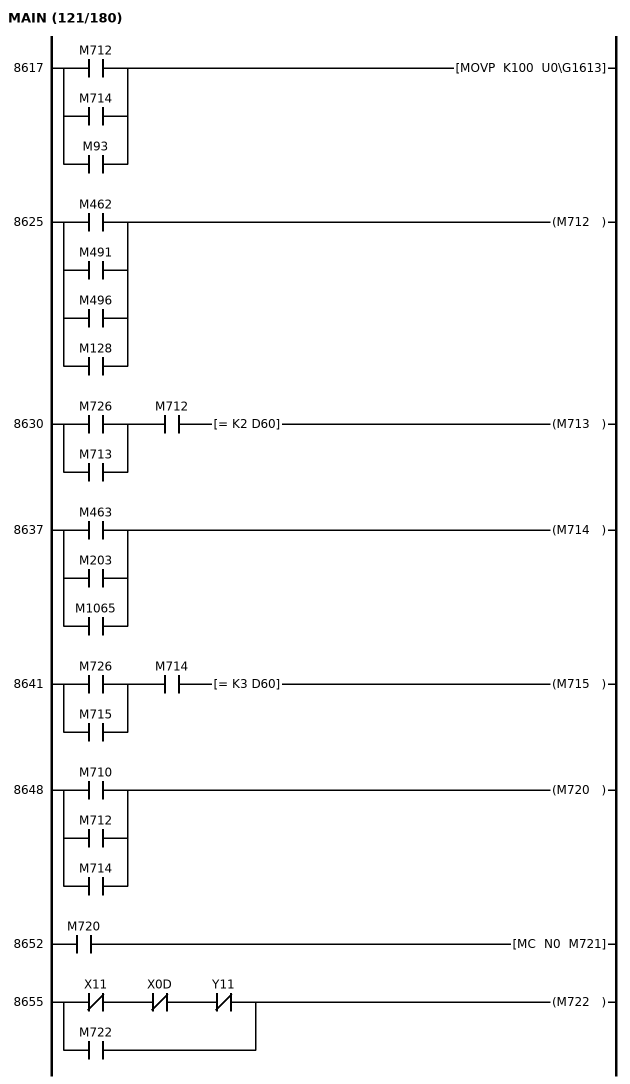
[picture p120: ladder of MAIN, rungs at steps 8617 to 8655]
8617  LD      M712
      OR      M714
      OR      M93
      MOVP    K100 U0\G1613
8625  LD      M462
      OR      M491
      OR      M496
      OR      M128
      OUT     M712
8630  LD      M726
      OR      M713
      AND     M712
      AND=    K2 D60
      OUT     M713
8637  LD      M463
      OR      M203
      OR      M1065
      OUT     M714
8641  LD      M726
      OR      M715
      AND     M714
      AND=    K3 D60
      OUT     M715
8648  LD      M710
      OR      M712
      OR      M714
      OUT     M720
8652  LD      M720
      MC      N0 M721
8655  LDI     X11
      ANI     X0D
      ANI     Y11
      OR      M722
      OUT     M722
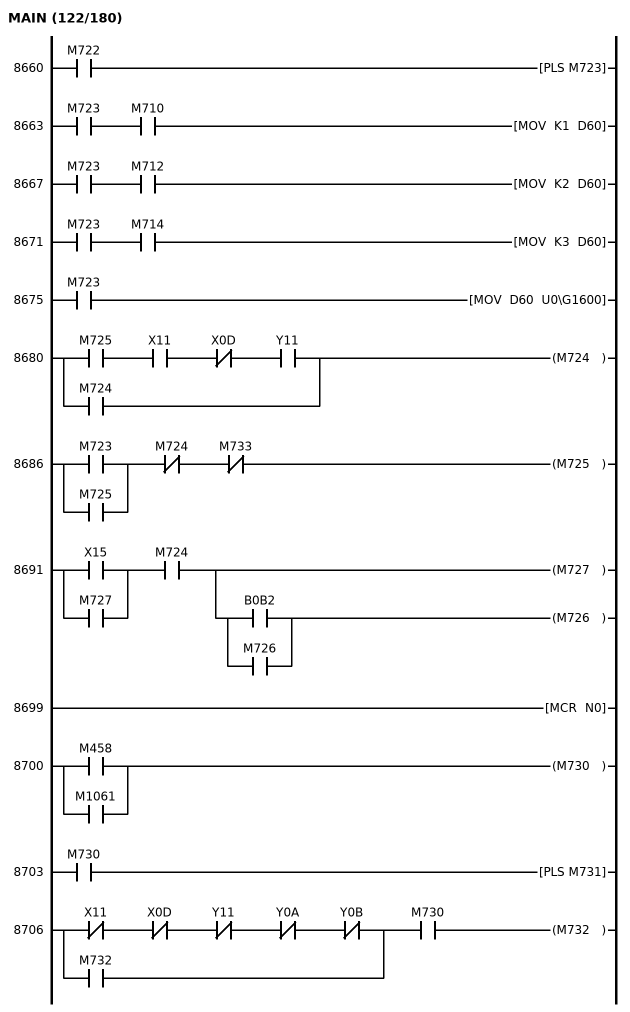
8660  LD      M722
      PLS     M723
8663  LD      M723
      AND     M710
      MOV     K1 D60
8667  LD      M723
      AND     M712
      MOV     K2 D60
8671  LD      M723
      AND     M714
      MOV     K3 D60
8675  LD      M723
      MOV     D60 U0\G1600
8680  LD      M725
      AND     X11
      ANI     X0D
      AND     Y11
      OR      M724
      OUT     M724
8686  LD      M723
      OR      M725
      ANI     M724
      ANI     M733
      OUT     M725
8691  LD      X15
      OR      M727
      AND     M724
      OUT     M727
      LD      B0B2
      OR      M726
      ANB
      OUT     M726
8699  MCR     N0
8700  LD      M458
      OR      M1061
      OUT     M730
8703  LD      M730
      PLS     M731
8706  LDI     X11
      ANI     X0D
      ANI     Y11
      ANI     Y0A
      ANI     Y0B
      OR      M732
      AND     M730
      OUT     M732
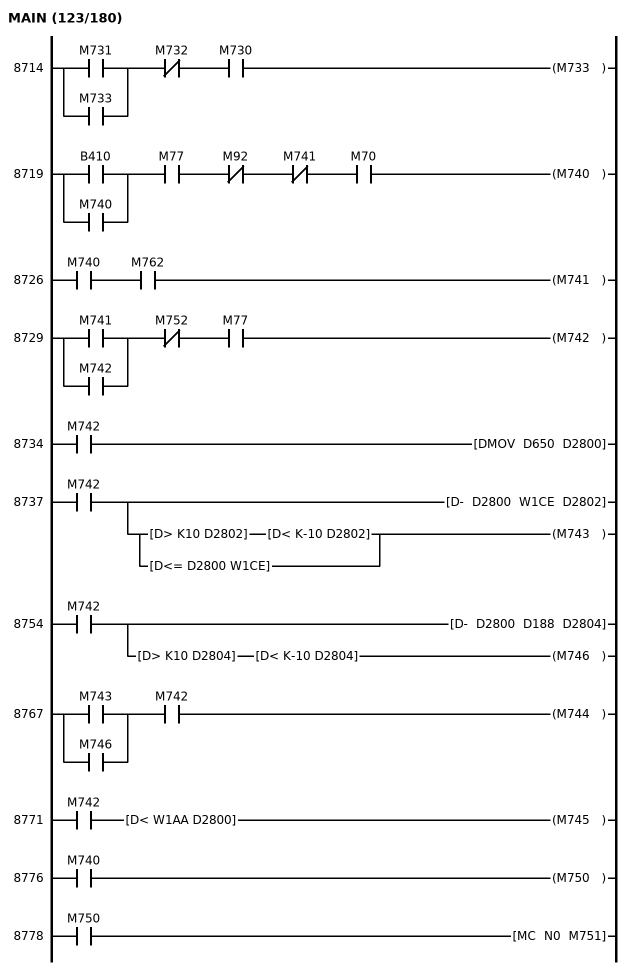
8714  LD      M731
      OR      M733
      ANI     M732
      AND     M730
      OUT     M733
8719  LD      B410
      OR      M740
      AND     M77
      ANI     M92
      ANI     M741
      AND     M70
      OUT     M740
8726  LD      M740
      AND     M762
      OUT     M741
8729  LD      M741
      OR      M742
      ANI     M752
      AND     M77
      OUT     M742
8734  LD      M742
      DMOV    D650 D2800
8737  LD      M742
      D-      D2800 W1CE D2802
      LDD>    K10 D2802
      ANDD<   K-10 D2802
      ORD<=   D2800 W1CE
      ANB
      OUT     M743
8754  LD      M742
      D-      D2800 D188 D2804
      ANDD>   K10 D2804
      ANDD<   K-10 D2804
      OUT     M746
8767  LD      M743
      OR      M746
      AND     M742
      OUT     M744
8771  LD      M742
      ANDD<   W1AA D2800
      OUT     M745
8776  LD      M740
      OUT     M750
8778  LD      M750
      MC      N0 M751
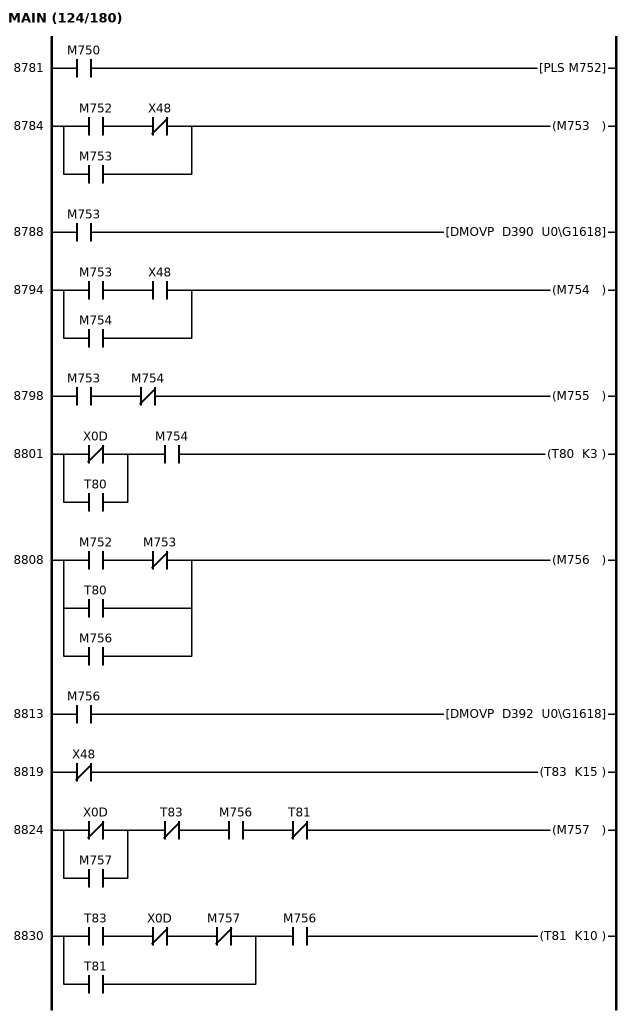
8781  LD      M750
      PLS     M752
8784  LD      M752
      ANI     X48
      OR      M753
      OUT     M753
8788  LD      M753
      DMOVP   D390 U0\G1618
8794  LD      M753
      AND     X48
      OR      M754
      OUT     M754
8798  LD      M753
      ANI     M754
      OUT     M755
8801  LDI     X0D
      OR      T80
      AND     M754
      OUT     T80 K3
8808  LD      M752
      ANI     M753
      OR      T80
      OR      M756
      OUT     M756
8813  LD      M756
      DMOVP   D392 U0\G1618
8819  LDI     X48
      OUT     T83 K15
8824  LDI     X0D
      OR      M757
      ANI     T83
      AND     M756
      ANI     T81
      OUT     M757
8830  LD      T83
      ANI     X0D
      ANI     M757
      OR      T81
      AND     M756
      OUT     T81 K10
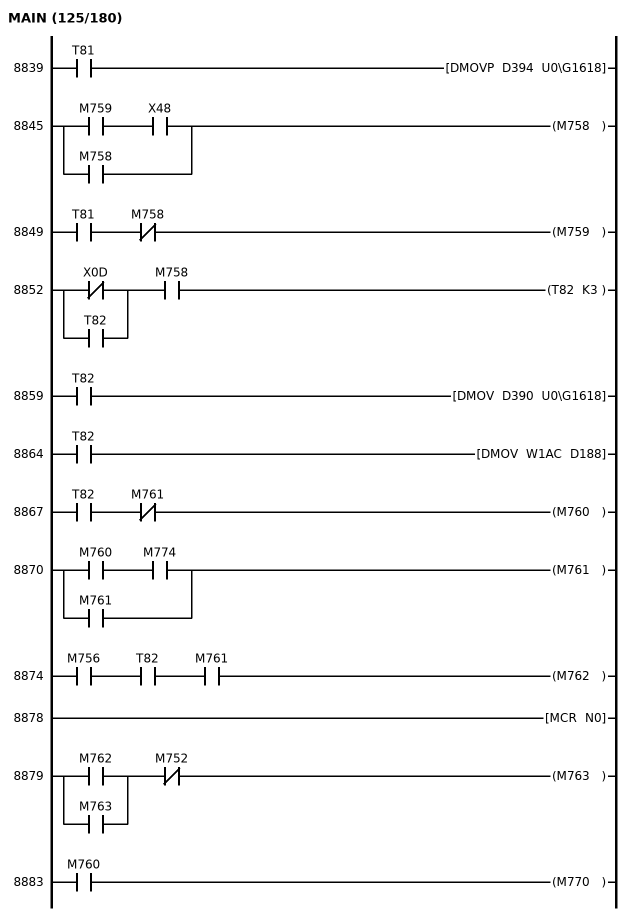
8839  LD      T81
      DMOVP   D394 U0\G1618
8845  LD      M759
      AND     X48
      OR      M758
      OUT     M758
8849  LD      T81
      ANI     M758
      OUT     M759
8852  LDI     X0D
      OR      T82
      AND     M758
      OUT     T82 K3
8859  LD      T82
      DMOV    D390 U0\G1618
8864  LD      T82
      DMOV    W1AC D188
8867  LD      T82
      ANI     M761
      OUT     M760
8870  LD      M760
      AND     M774
      OR      M761
      OUT     M761
8874  LD      M756
      AND     T82
      AND     M761
      OUT     M762
8878  MCR     N0
8879  LD      M762
      OR      M763
      ANI     M752
      OUT     M763
8883  LD      M760
      OUT     M770
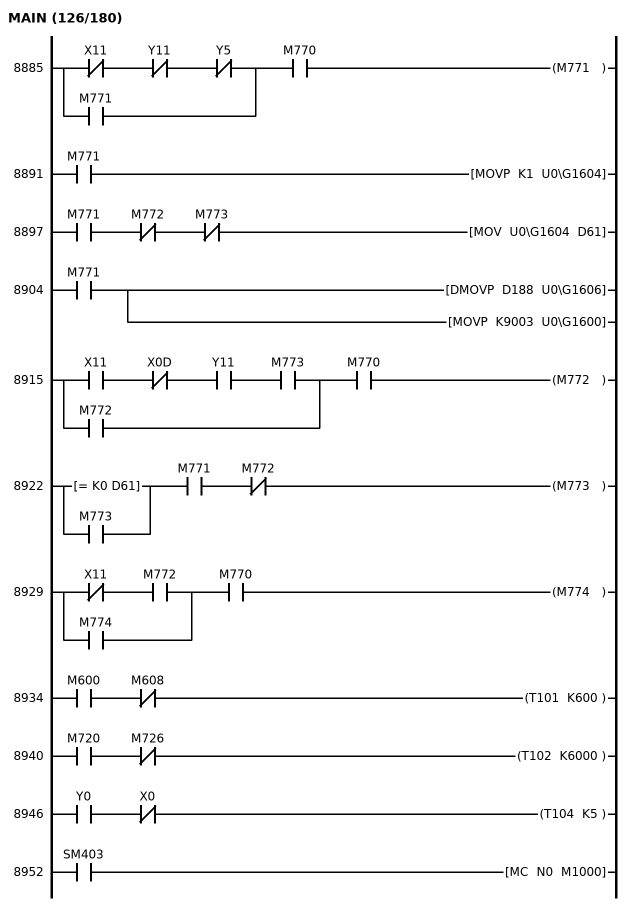
8885  LDI     X11
      ANI     Y11
      ANI     Y5
      OR      M771
      AND     M770
      OUT     M771
8891  LD      M771
      MOVP    K1 U0\G1604
8897  LD      M771
      ANI     M772
      ANI     M773
      MOV     U0\G1604 D61
8904  LD      M771
      DMOVP   D188 U0\G1606
      MOVP    K9003 U0\G1600
8915  LD      X11
      ANI     X0D
      AND     Y11
      AND     M773
      OR      M772
      AND     M770
      OUT     M772
8922  LD=     K0 D61
      OR      M773
      AND     M771
      ANI     M772
      OUT     M773
8929  LDI     X11
      AND     M772
      OR      M774
      AND     M770
      OUT     M774
8934  LD      M600
      ANI     M608
      OUT     T101 K600
8940  LD      M720
      ANI     M726
      OUT     T102 K6000
8946  LD      Y0
      ANI     X0
      OUT     T104 K5
8952  LD      SM403
      MC      N0 M1000
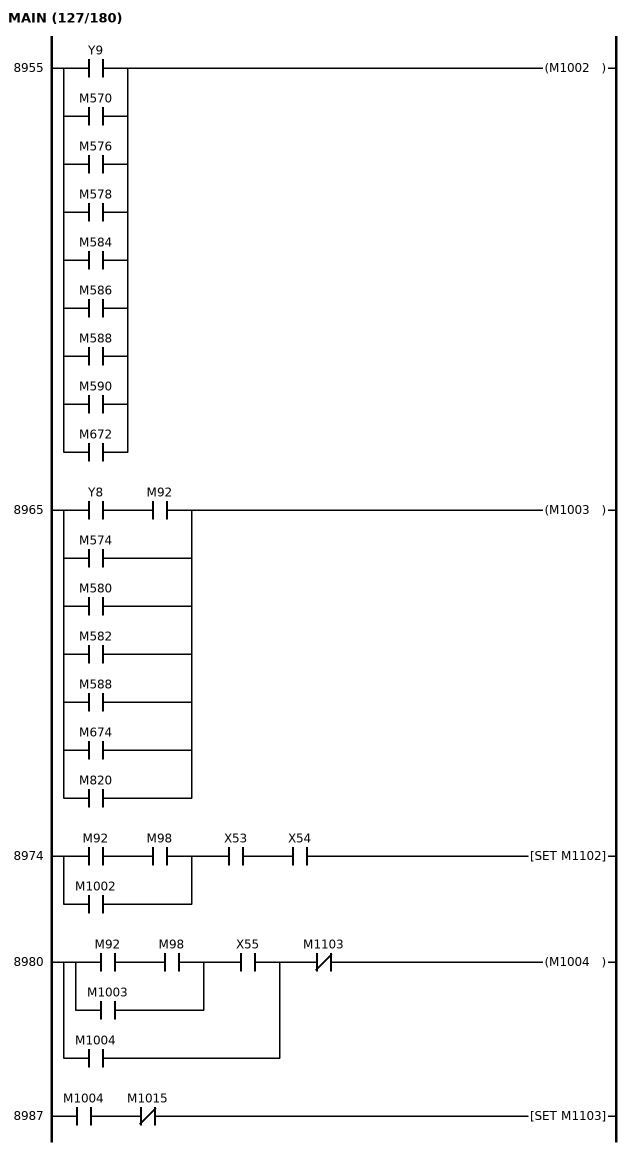
8955  LD      Y9
      OR      M570
      OR      M576
      OR      M578
      OR      M584
      OR      M586
      OR      M588
      OR      M590
      OR      M672
      OUT     M1002
8965  LD      Y8
      AND     M92
      OR      M574
      OR      M580
      OR      M582
      OR      M588
      OR      M674
      OR      M820
      OUT     M1003
8974  LD      M92
      AND     M98
      OR      M1002
      AND     X53
      AND     X54
      SET     M1102
8980  LD      M92
      AND     M98
      OR      M1003
      AND     X55
      OR      M1004
      ANI     M1103
      OUT     M1004
8987  LD      M1004
      ANI     M1015
      SET     M1103
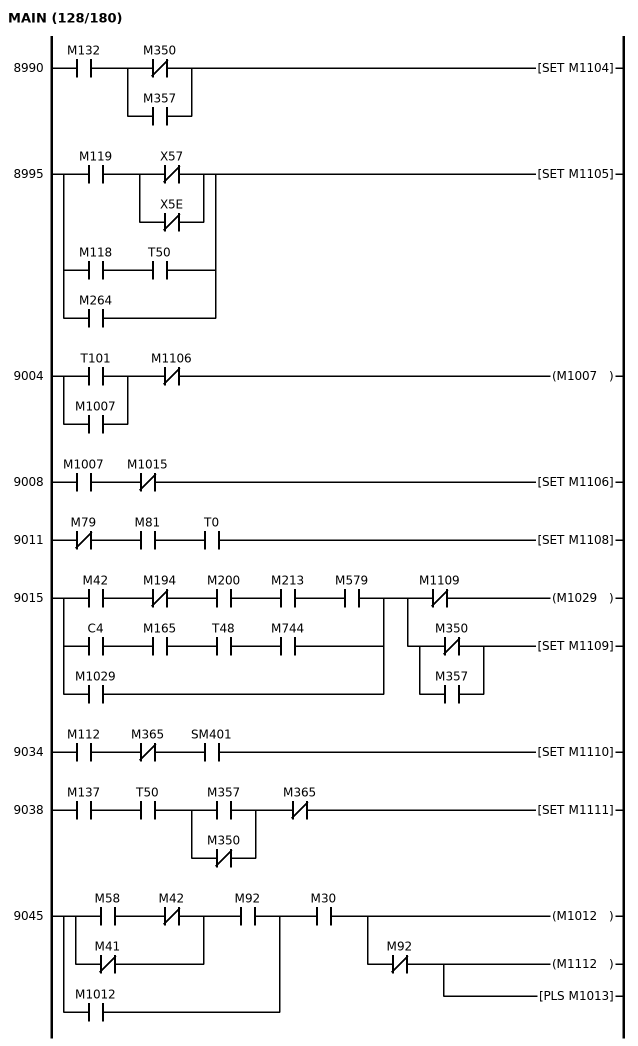
8990  LD      M132
      LDI     M350
      OR      M357
      ANB
      SET     M1104
8995  LD      M119
      LDI     X57
      ORI     X5E
      ANB
      LD      M118
      AND     T50
      ORB
      OR      M264
      SET     M1105
9004  LD      T101
      OR      M1007
      ANI     M1106
      OUT     M1007
9008  LD      M1007
      ANI     M1015
      SET     M1106
9011  LDI     M79
      AND     M81
      AND     T0
      SET     M1108
9015  LD      M42
      ANI     M194
      AND     M200
      AND     M213
      AND     M579
      LD      C4
      AND     M165
      AND     T48
      AND     M744
      ORB
      OR      M1029
      MPS
      ANI     M1109
      OUT     M1029
      MPP
      LDI     M350
      OR      M357
      ANB
      SET     M1109
9034  LD      M112
      ANI     M365
      AND     SM401
      SET     M1110
9038  LD      M137
      AND     T50
      LD      M357
      ORI     M350
      ANB
      ANI     M365
      SET     M1111
9045  LD      M58
      ANI     M42
      ORI     M41
      AND     M92
      OR      M1012
      AND     M30
      OUT     M1012
      ANI     M92
      OUT     M1112
      PLS     M1013
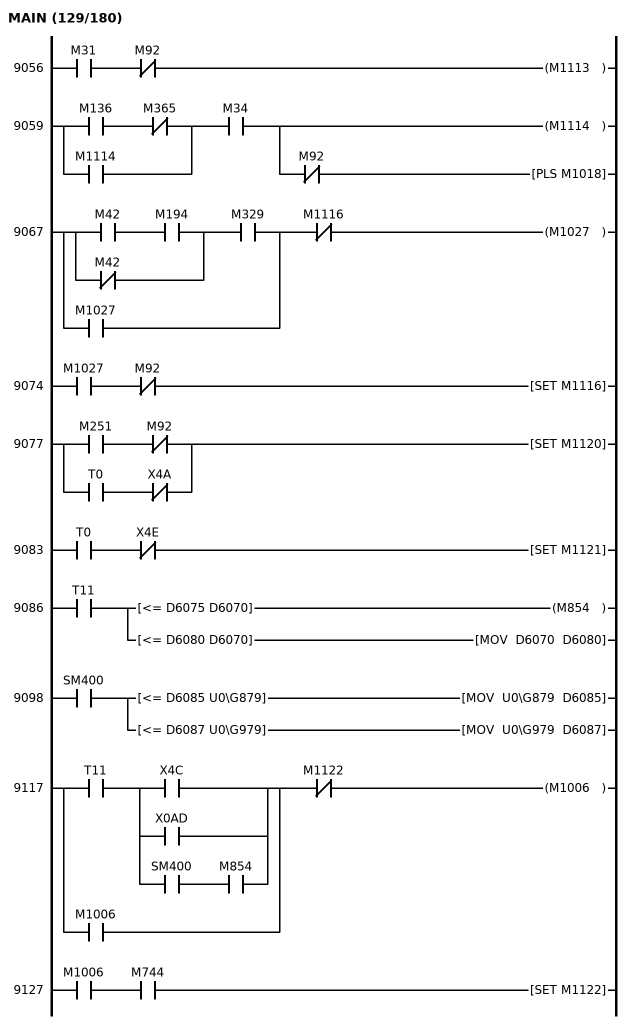
9056  LD      M31
      ANI     M92
      OUT     M1113
9059  LD      M136
      ANI     M365
      OR      M1114
      AND     M34
      OUT     M1114
      ANI     M92
      PLS     M1018
9067  LD      M42
      AND     M194
      ORI     M42
      AND     M329
      OR      M1027
      ANI     M1116
      OUT     M1027
9074  LD      M1027
      ANI     M92
      SET     M1116
9077  LD      M251
      ANI     M92
      LD      T0
      ANI     X4A
      ORB
      SET     M1120
9083  LD      T0
      ANI     X4E
      SET     M1121
9086  LD      T11
      MPS
      AND<=   D6075 D6070
      OUT     M854
      MPP
      AND<=   D6080 D6070
      MOV     D6070 D6080
9098  LD      SM400
      MPS
      AND<=   D6085 U0\G879
      MOV     U0\G879 D6085
      MPP
      AND<=   D6087 U0\G979
      MOV     U0\G979 D6087
9117  LD      T11
      LD      X4C
      OR      X0AD
      LD      SM400
      AND     M854
      ORB
      ANB
      OR      M1006
      ANI     M1122
      OUT     M1006
9127  LD      M1006
      AND     M744
      SET     M1122
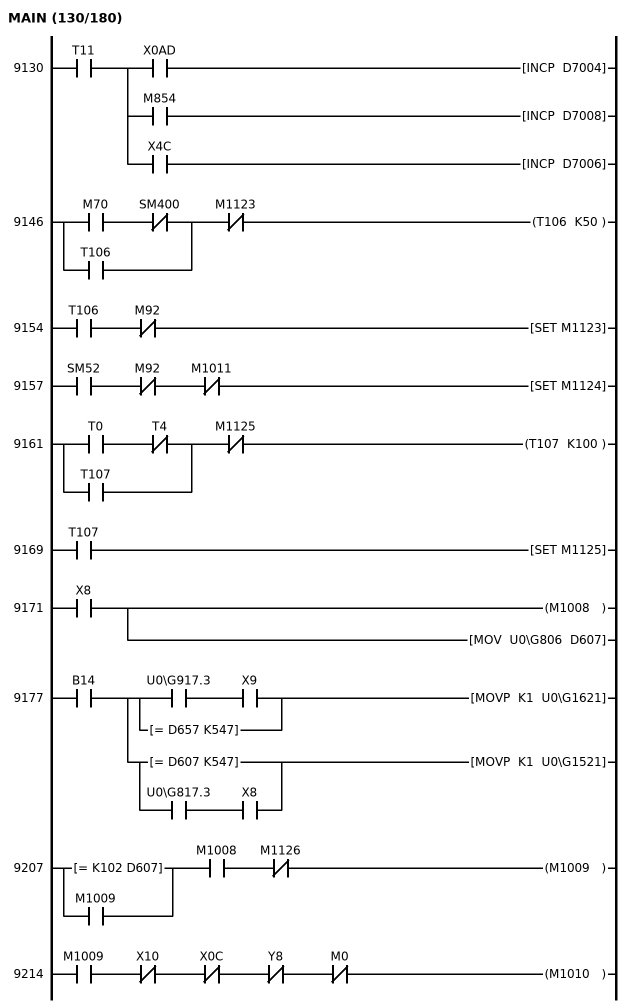
9130  LD      T11
      MPS
      AND     X0AD
      INCP    D7004
      MRD
      AND     M854
      INCP    D7008
      MPP
      AND     X4C
      INCP    D7006
9146  LD      M70
      ANI     SM400
      OR      T106
      ANI     M1123
      OUT     T106 K50
9154  LD      T106
      ANI     M92
      SET     M1123
9157  LD      SM52
      ANI     M92
      ANI     M1011
      SET     M1124
9161  LD      T0
      ANI     T4
      OR      T107
      ANI     M1125
      OUT     T107 K100
9169  LD      T107
      SET     M1125
9171  LD      X8
      OUT     M1008
      MOV     U0\G806 D607
9177  LD      B14
      MPS
      LD      U0\G917.3
      AND     X9
      OR=     D657 K547
      ANB
      MOVP    K1 U0\G1621
      MPP
      LD=     D607 K547
      LD      U0\G817.3
      AND     X8
      ORB
      ANB
      MOVP    K1 U0\G1521
9207  LD=     K102 D607
      OR      M1009
      AND     M1008
      ANI     M1126
      OUT     M1009
9214  LD      M1009
      ANI     X10
      ANI     X0C
      ANI     Y8
      ANI     M0
      OUT     M1010
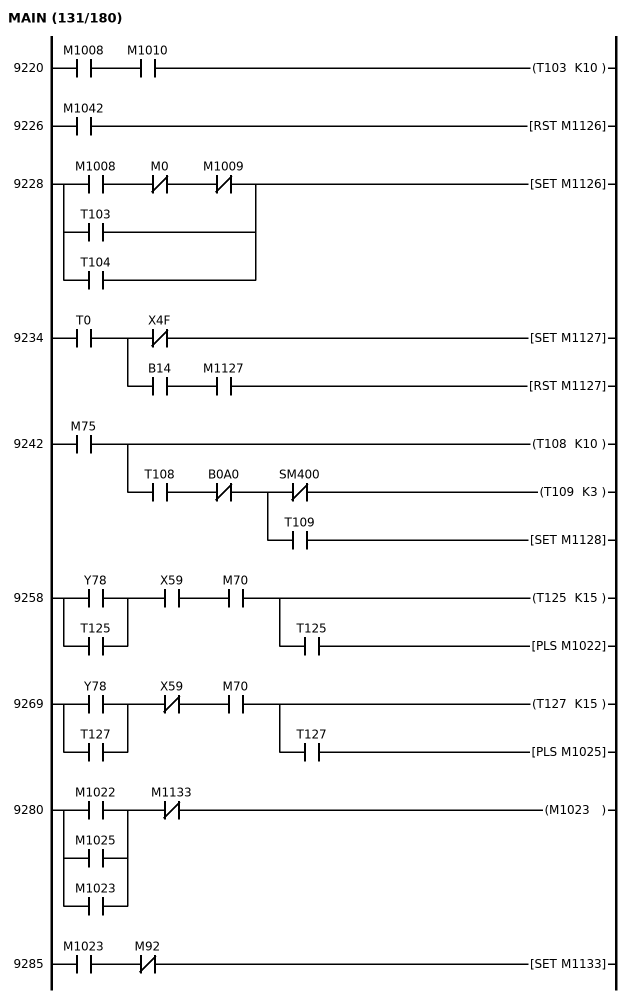
9220  LD      M1008
      AND     M1010
      OUT     T103 K10
9226  LD      M1042
      RST     M1126
9228  LD      M1008
      ANI     M0
      ANI     M1009
      OR      T103
      OR      T104
      SET     M1126
9234  LD      T0
      MPS
      ANI     X4F
      SET     M1127
      MPP
      AND     B14
      AND     M1127
      RST     M1127
9242  LD      M75
      OUT     T108 K10
      AND     T108
      ANI     B0A0
      MPS
      ANI     SM400
      OUT     T109 K3
      MPP
      AND     T109
      SET     M1128
9258  LD      Y78
      OR      T125
      AND     X59
      AND     M70
      OUT     T125 K15
      AND     T125
      PLS     M1022
9269  LD      Y78
      OR      T127
      ANI     X59
      AND     M70
      OUT     T127 K15
      AND     T127
      PLS     M1025
9280  LD      M1022
      OR      M1025
      OR      M1023
      ANI     M1133
      OUT     M1023
9285  LD      M1023
      ANI     M92
      SET     M1133
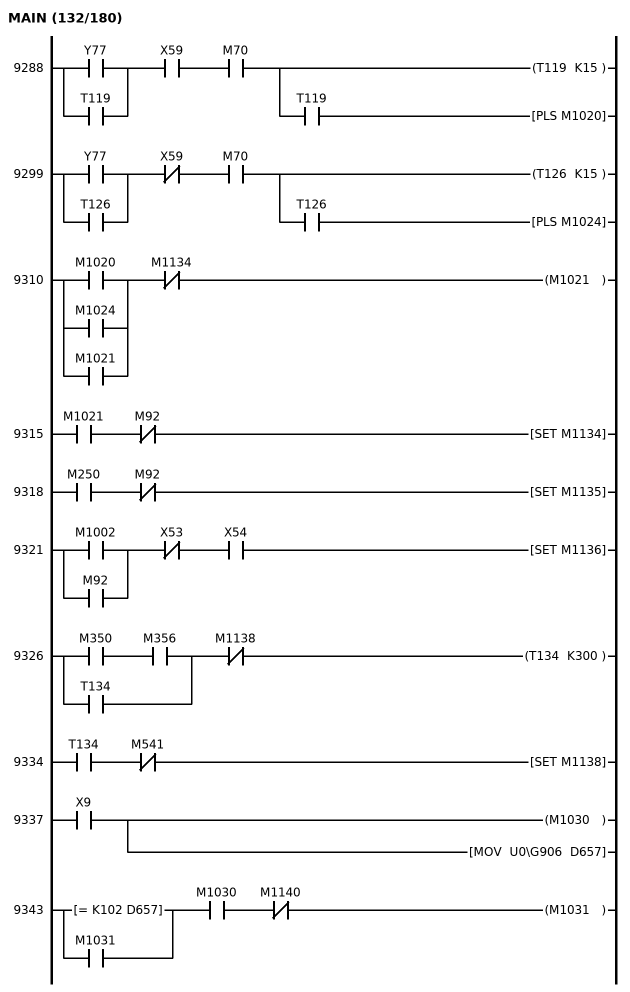
9288  LD      Y77
      OR      T119
      AND     X59
      AND     M70
      OUT     T119 K15
      AND     T119
      PLS     M1020
9299  LD      Y77
      OR      T126
      ANI     X59
      AND     M70
      OUT     T126 K15
      AND     T126
      PLS     M1024
9310  LD      M1020
      OR      M1024
      OR      M1021
      ANI     M1134
      OUT     M1021
9315  LD      M1021
      ANI     M92
      SET     M1134
9318  LD      M250
      ANI     M92
      SET     M1135
9321  LD      M1002
      OR      M92
      ANI     X53
      AND     X54
      SET     M1136
9326  LD      M350
      AND     M356
      OR      T134
      ANI     M1138
      OUT     T134 K300
9334  LD      T134
      ANI     M541
      SET     M1138
9337  LD      X9
      OUT     M1030
      MOV     U0\G906 D657
9343  LD=     K102 D657
      OR      M1031
      AND     M1030
      ANI     M1140
      OUT     M1031
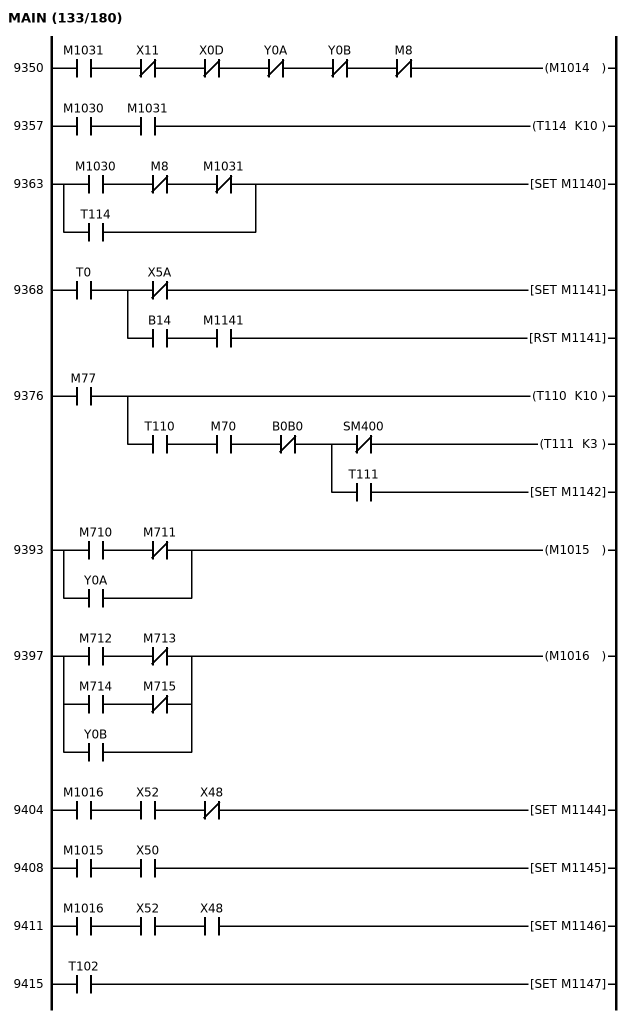
9350  LD      M1031
      ANI     X11
      ANI     X0D
      ANI     Y0A
      ANI     Y0B
      ANI     M8
      OUT     M1014
9357  LD      M1030
      AND     M1031
      OUT     T114 K10
9363  LD      M1030
      ANI     M8
      ANI     M1031
      OR      T114
      SET     M1140
9368  LD      T0
      MPS
      ANI     X5A
      SET     M1141
      MPP
      AND     B14
      AND     M1141
      RST     M1141
9376  LD      M77
      OUT     T110 K10
      AND     T110
      AND     M70
      ANI     B0B0
      MPS
      ANI     SM400
      OUT     T111 K3
      MPP
      AND     T111
      SET     M1142
9393  LD      M710
      ANI     M711
      OR      Y0A
      OUT     M1015
9397  LD      M712
      ANI     M713
      LD      M714
      ANI     M715
      ORB
      OR      Y0B
      OUT     M1016
9404  LD      M1016
      AND     X52
      ANI     X48
      SET     M1144
9408  LD      M1015
      AND     X50
      SET     M1145
9411  LD      M1016
      AND     X52
      AND     X48
      SET     M1146
9415  LD      T102
      SET     M1147
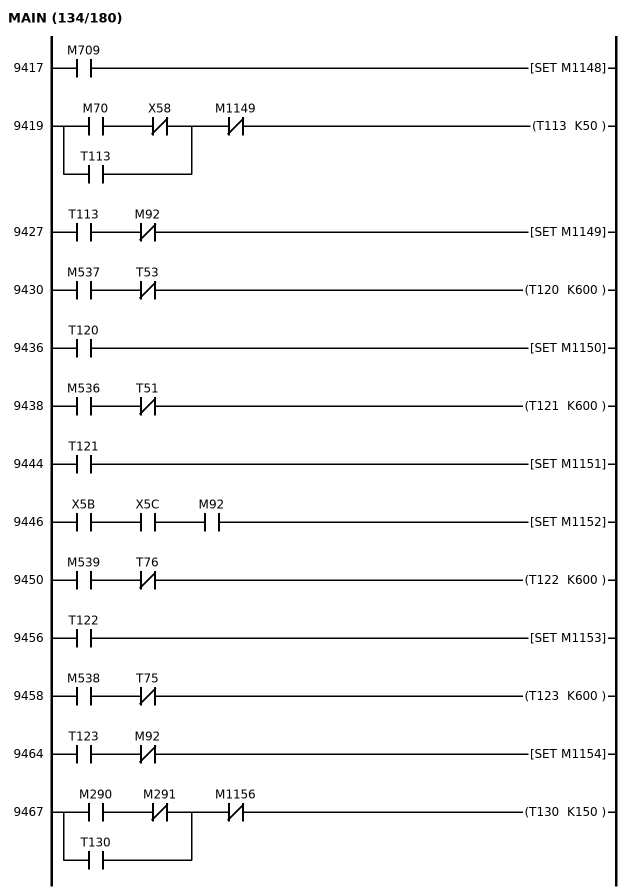
9417  LD      M709
      SET     M1148
9419  LD      M70
      ANI     X58
      OR      T113
      ANI     M1149
      OUT     T113 K50
9427  LD      T113
      ANI     M92
      SET     M1149
9430  LD      M537
      ANI     T53
      OUT     T120 K600
9436  LD      T120
      SET     M1150
9438  LD      M536
      ANI     T51
      OUT     T121 K600
9444  LD      T121
      SET     M1151
9446  LD      X5B
      AND     X5C
      AND     M92
      SET     M1152
9450  LD      M539
      ANI     T76
      OUT     T122 K600
9456  LD      T122
      SET     M1153
9458  LD      M538
      ANI     T75
      OUT     T123 K600
9464  LD      T123
      ANI     M92
      SET     M1154
9467  LD      M290
      ANI     M291
      OR      T130
      ANI     M1156
      OUT     T130 K150
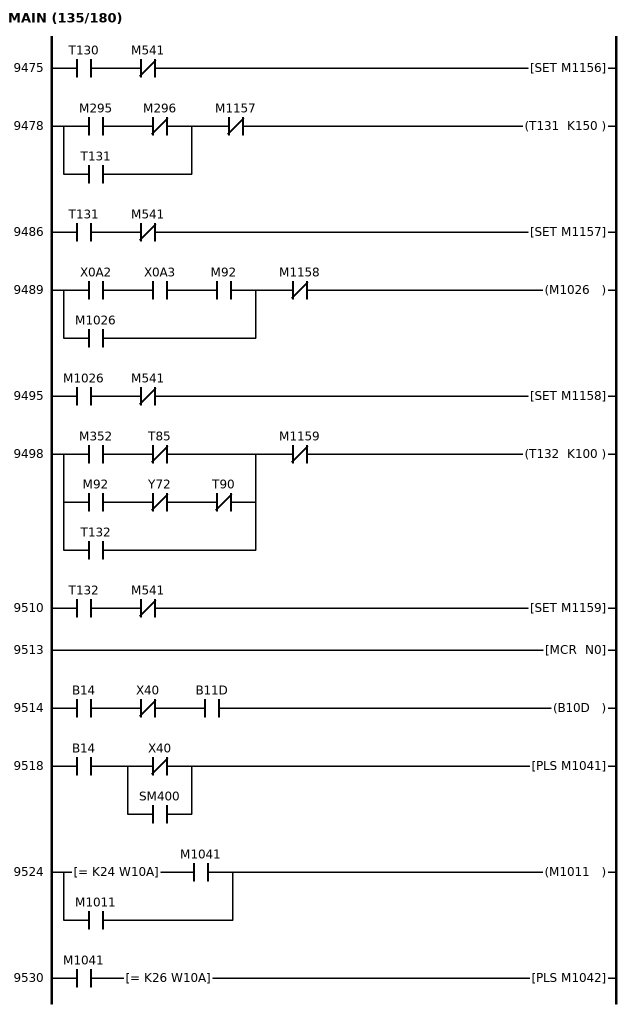
9475  LD      T130
      ANI     M541
      SET     M1156
9478  LD      M295
      ANI     M296
      OR      T131
      ANI     M1157
      OUT     T131 K150
9486  LD      T131
      ANI     M541
      SET     M1157
9489  LD      X0A2
      AND     X0A3
      AND     M92
      OR      M1026
      ANI     M1158
      OUT     M1026
9495  LD      M1026
      ANI     M541
      SET     M1158
9498  LD      M352
      ANI     T85
      LD      M92
      ANI     Y72
      ANI     T90
      ORB
      OR      T132
      ANI     M1159
      OUT     T132 K100
9510  LD      T132
      ANI     M541
      SET     M1159
9513  MCR     N0
9514  LD      B14
      ANI     X40
      AND     B11D
      OUT     B10D
9518  LD      B14
      LDI     X40
      OR      SM400
      ANB
      PLS     M1041
9524  LD=     K24 W10A
      AND     M1041
      OR      M1011
      OUT     M1011
9530  LD      M1041
      AND=    K26 W10A
      PLS     M1042
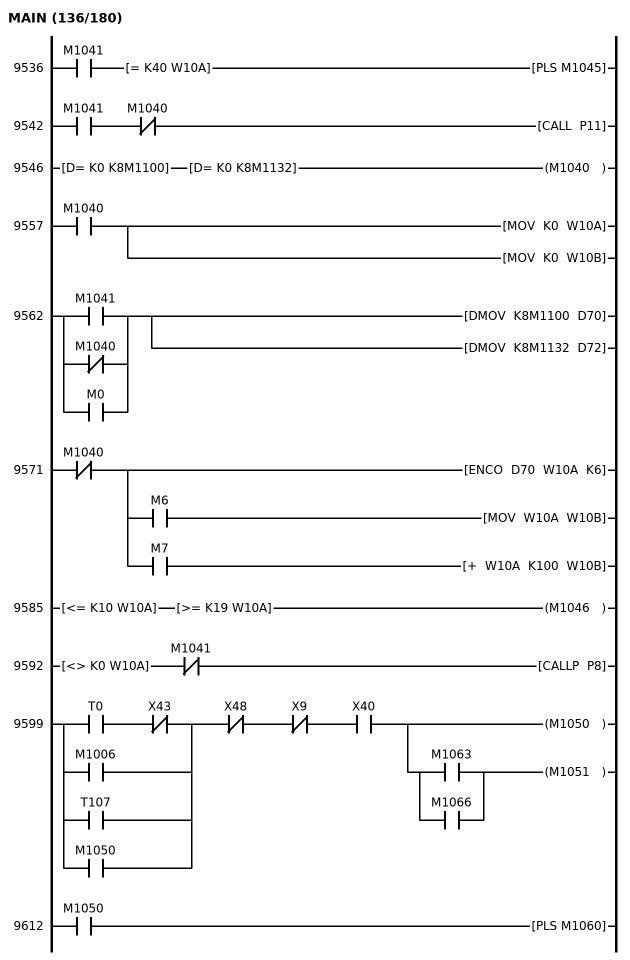
9536  LD      M1041
      AND=    K40 W10A
      PLS     M1045
9542  LD      M1041
      ANI     M1040
      CALL    P11
9546  LDD=    K0 K8M1100
      ANDD=   K0 K8M1132
      OUT     M1040
9557  LD      M1040
      MOV     K0 W10A
      MOV     K0 W10B
9562  LD      M1041
      ORI     M1040
      OR      M0
      DMOV    K8M1100 D70
      DMOV    K8M1132 D72
9571  LDI     M1040
      ENCO    D70 W10A K6
      MPS
      AND     M6
      MOV     W10A W10B
      MPP
      AND     M7
      +       W10A K100 W10B
9585  LD<=    K10 W10A
      AND>=   K19 W10A
      OUT     M1046
9592  LD<>    K0 W10A
      ANI     M1041
      CALLP   P8
9599  LD      T0
      ANI     X43
      OR      M1006
      OR      T107
      OR      M1050
      ANI     X48
      ANI     X9
      AND     X40
      OUT     M1050
      LD      M1063
      OR      M1066
      ANB
      OUT     M1051
9612  LD      M1050
      PLS     M1060
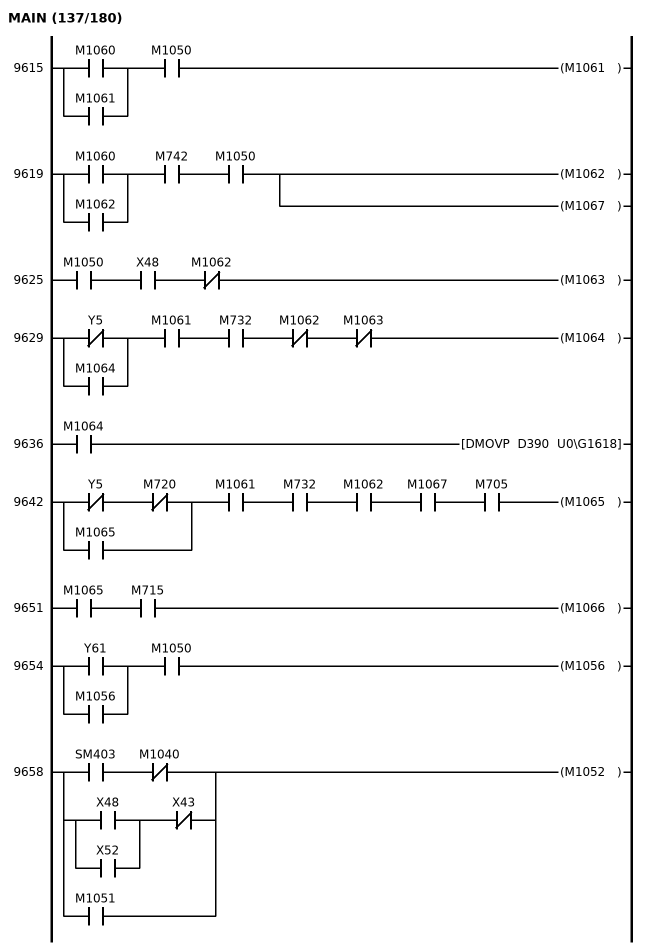
9615  LD      M1060
      OR      M1061
      AND     M1050
      OUT     M1061
9619  LD      M1060
      OR      M1062
      AND     M742
      AND     M1050
      OUT     M1062
      OUT     M1067
9625  LD      M1050
      AND     X48
      ANI     M1062
      OUT     M1063
9629  LDI     Y5
      OR      M1064
      AND     M1061
      AND     M732
      ANI     M1062
      ANI     M1063
      OUT     M1064
9636  LD      M1064
      DMOVP   D390 U0\G1618
9642  LDI     Y5
      ANI     M720
      OR      M1065
      AND     M1061
      AND     M732
      AND     M1062
      AND     M1067
      AND     M705
      OUT     M1065
9651  LD      M1065
      AND     M715
      OUT     M1066
9654  LD      Y61
      OR      M1056
      AND     M1050
      OUT     M1056
9658  LD      SM403
      ANI     M1040
      LD      X48
      OR      X52
      ANI     X43
      ORB
      OR      M1051
      OUT     M1052
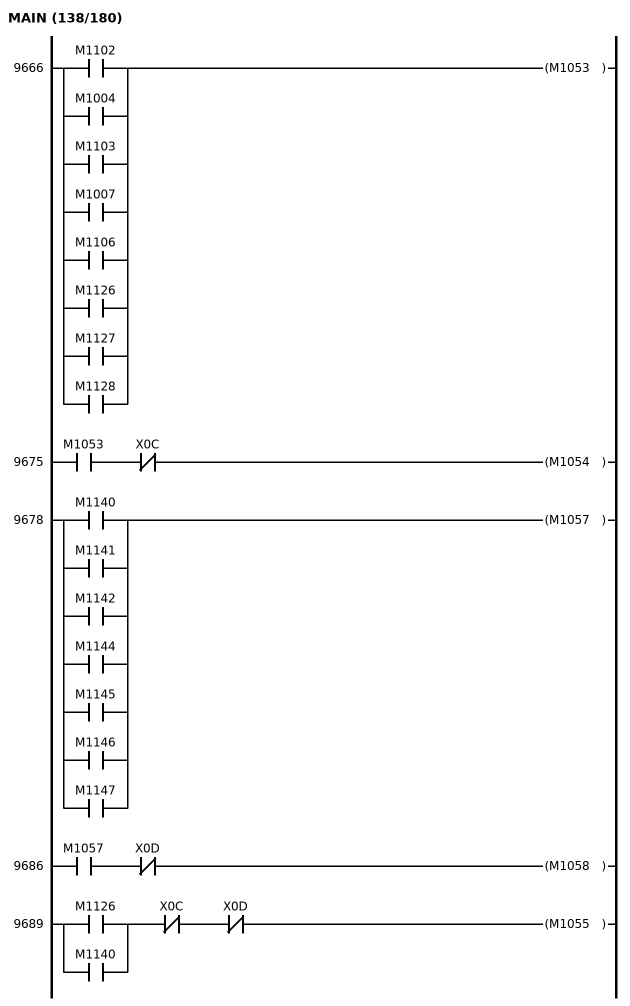
9666  LD      M1102
      OR      M1004
      OR      M1103
      OR      M1007
      OR      M1106
      OR      M1126
      OR      M1127
      OR      M1128
      OUT     M1053
9675  LD      M1053
      ANI     X0C
      OUT     M1054
9678  LD      M1140
      OR      M1141
      OR      M1142
      OR      M1144
      OR      M1145
      OR      M1146
      OR      M1147
      OUT     M1057
9686  LD      M1057
      ANI     X0D
      OUT     M1058
9689  LD      M1126
      OR      M1140
      ANI     X0C
      ANI     X0D
      OUT     M1055
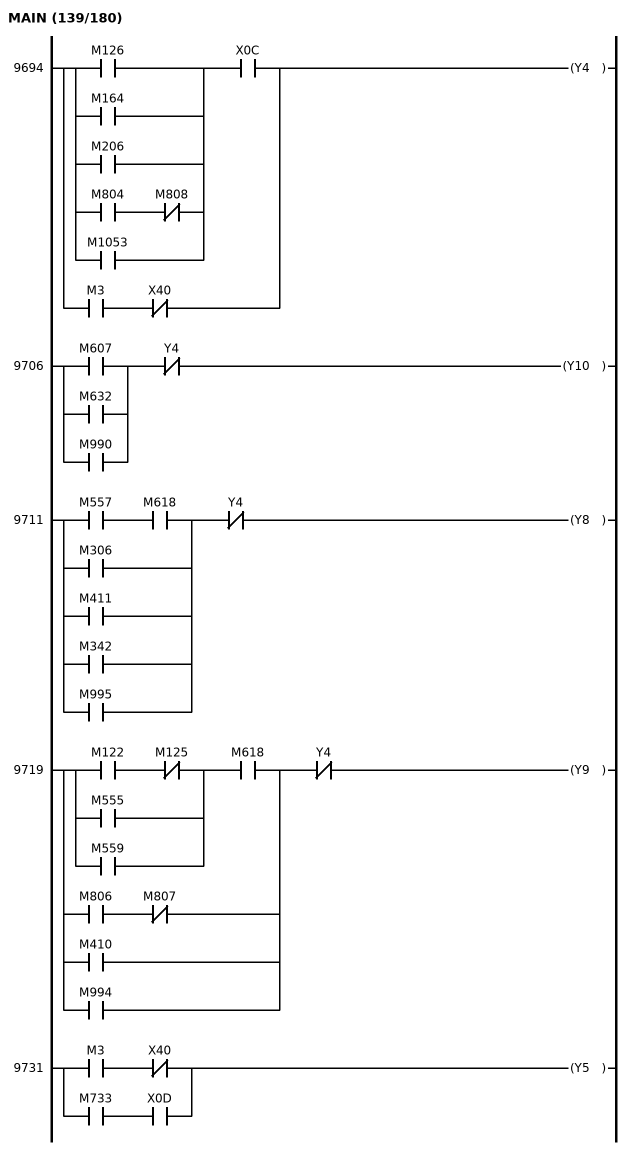
9694  LD      M126
      OR      M164
      OR      M206
      LD      M804
      ANI     M808
      ORB
      OR      M1053
      AND     X0C
      LD      M3
      ANI     X40
      ORB
      OUT     Y4
9706  LD      M607
      OR      M632
      OR      M990
      ANI     Y4
      OUT     Y10
9711  LD      M557
      AND     M618
      OR      M306
      OR      M411
      OR      M342
      OR      M995
      ANI     Y4
      OUT     Y8
9719  LD      M122
      ANI     M125
      OR      M555
      OR      M559
      AND     M618
      LD      M806
      ANI     M807
      ORB
      OR      M410
      OR      M994
      ANI     Y4
      OUT     Y9
9731  LD      M3
      ANI     X40
      LD      M733
      AND     X0D
      ORB
      OUT     Y5
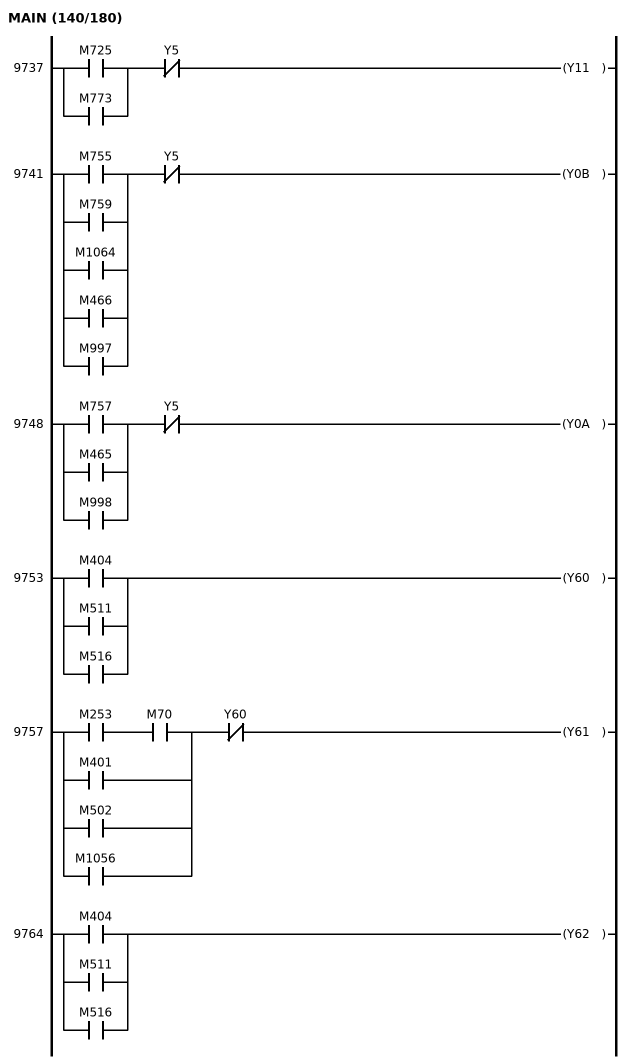
9737  LD      M725
      OR      M773
      ANI     Y5
      OUT     Y11
9741  LD      M755
      OR      M759
      OR      M1064
      OR      M466
      OR      M997
      ANI     Y5
      OUT     Y0B
9748  LD      M757
      OR      M465
      OR      M998
      ANI     Y5
      OUT     Y0A
9753  LD      M404
      OR      M511
      OR      M516
      OUT     Y60
9757  LD      M253
      AND     M70
      OR      M401
      OR      M502
      OR      M1056
      ANI     Y60
      OUT     Y61
9764  LD      M404
      OR      M511
      OR      M516
      OUT     Y62
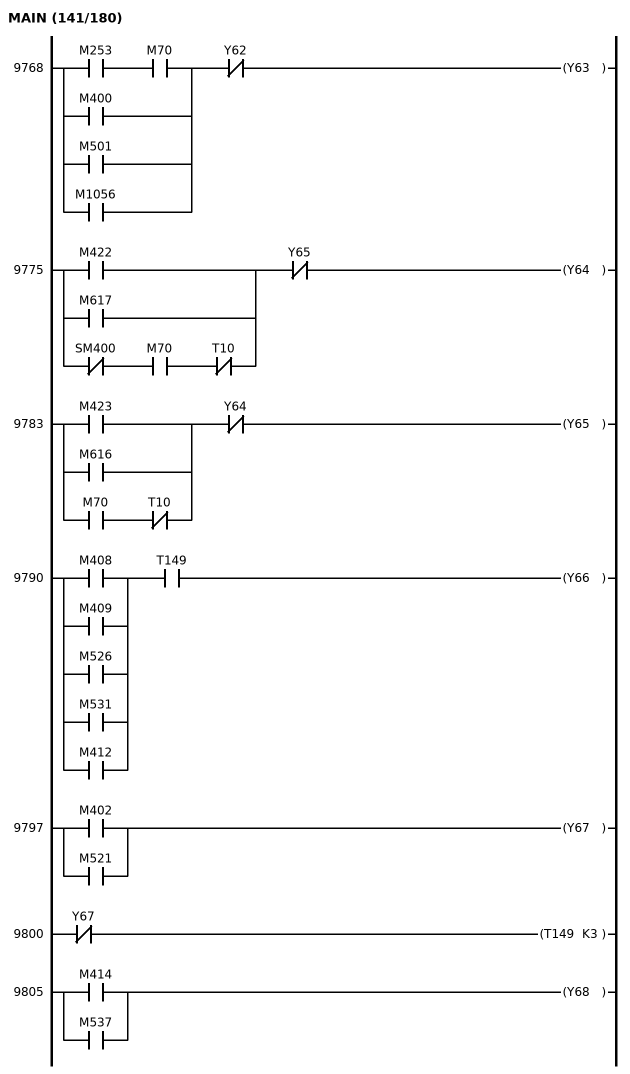
9768  LD      M253
      AND     M70
      OR      M400
      OR      M501
      OR      M1056
      ANI     Y62
      OUT     Y63
9775  LD      M422
      OR      M617
      LDI     SM400
      AND     M70
      ANI     T10
      ORB
      ANI     Y65
      OUT     Y64
9783  LD      M423
      OR      M616
      LD      M70
      ANI     T10
      ORB
      ANI     Y64
      OUT     Y65
9790  LD      M408
      OR      M409
      OR      M526
      OR      M531
      OR      M412
      AND     T149
      OUT     Y66
9797  LD      M402
      OR      M521
      OUT     Y67
9800  LDI     Y67
      OUT     T149 K3
9805  LD      M414
      OR      M537
      OUT     Y68
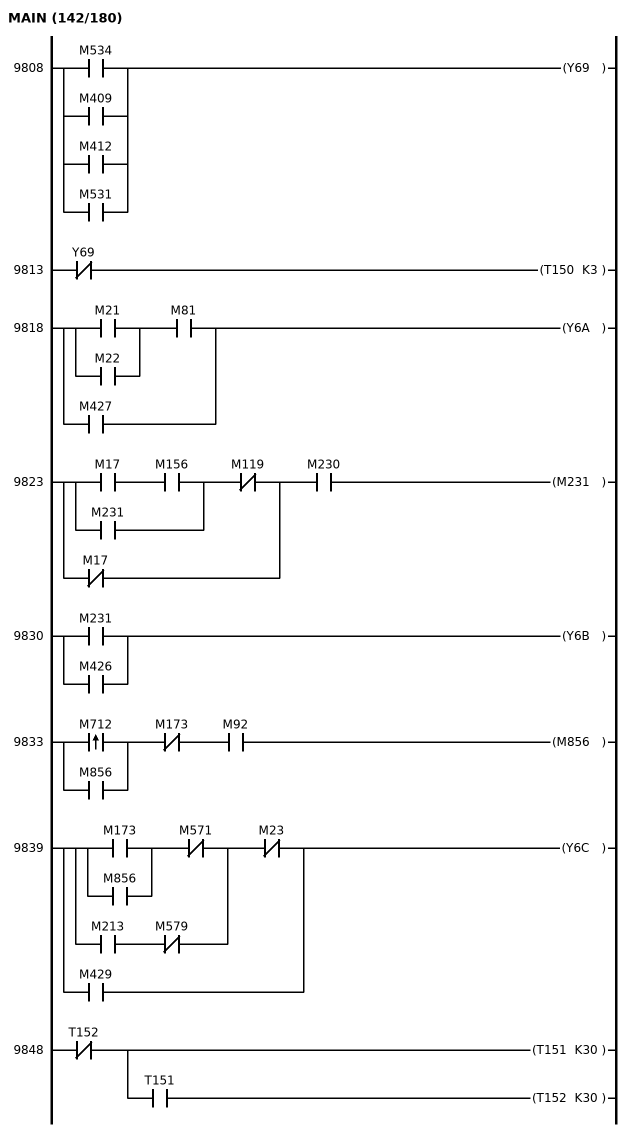
9808  LD      M534
      OR      M409
      OR      M412
      OR      M531
      OUT     Y69
9813  LDI     Y69
      OUT     T150 K3
9818  LD      M21
      OR      M22
      AND     M81
      OR      M427
      OUT     Y6A
9823  LD      M17
      AND     M156
      OR      M231
      ANI     M119
      ORI     M17
      AND     M230
      OUT     M231
9830  LD      M231
      OR      M426
      OUT     Y6B
9833  LDP     M712
      OR      M856
      ANI     M173
      AND     M92
      OUT     M856
9839  LD      M173
      OR      M856
      ANI     M571
      LD      M213
      ANI     M579
      ORB
      ANI     M23
      OR      M429
      OUT     Y6C
9848  LDI     T152
      OUT     T151 K30
      AND     T151
      OUT     T152 K30
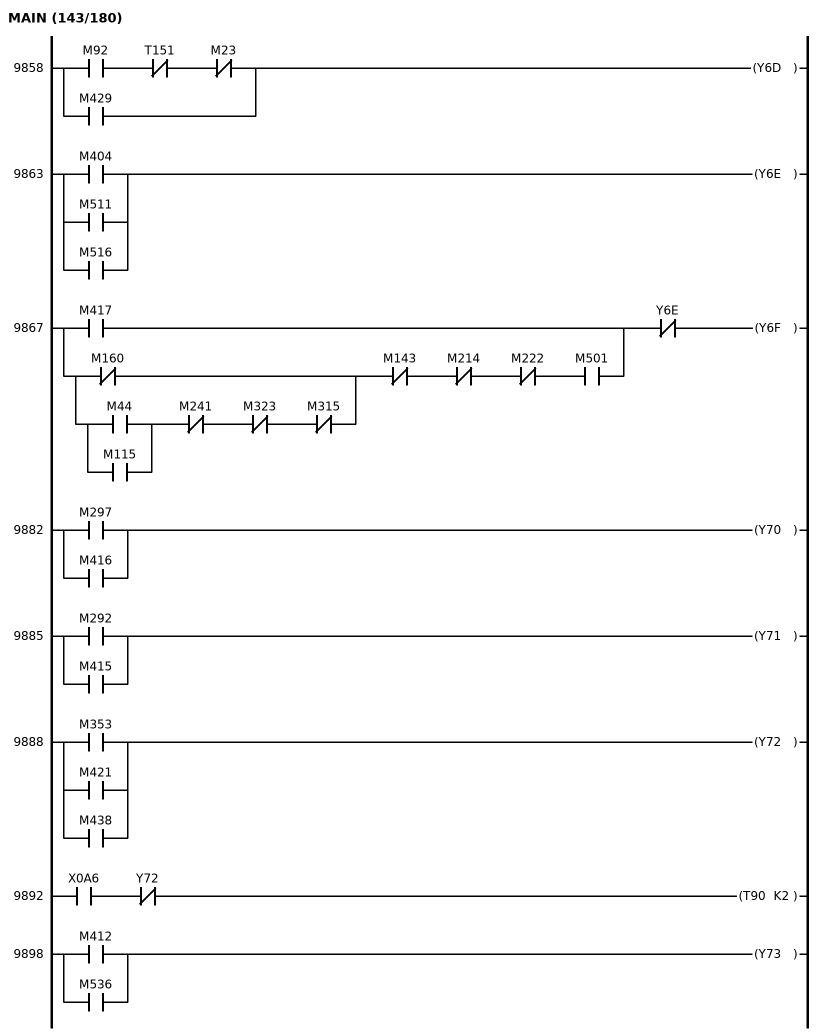
9858  LD      M92
      ANI     T151
      ANI     M23
      OR      M429
      OUT     Y6D
9863  LD      M404
      OR      M511
      OR      M516
      OUT     Y6E
9867  LD      M417
      LDI     M160
      LD      M44
      OR      M115
      ANI     M241
      ANI     M323
      ANI     M315
      ORB
      ANI     M143
      ANI     M214
      ANI     M222
      AND     M501
      ORB
      ANI     Y6E
      OUT     Y6F
9882  LD      M297
      OR      M416
      OUT     Y70
9885  LD      M292
      OR      M415
      OUT     Y71
9888  LD      M353
      OR      M421
      OR      M438
      OUT     Y72
9892  LD      X0A6
      ANI     Y72
      OUT     T90 K2
9898  LD      M412
      OR      M536
      OUT     Y73
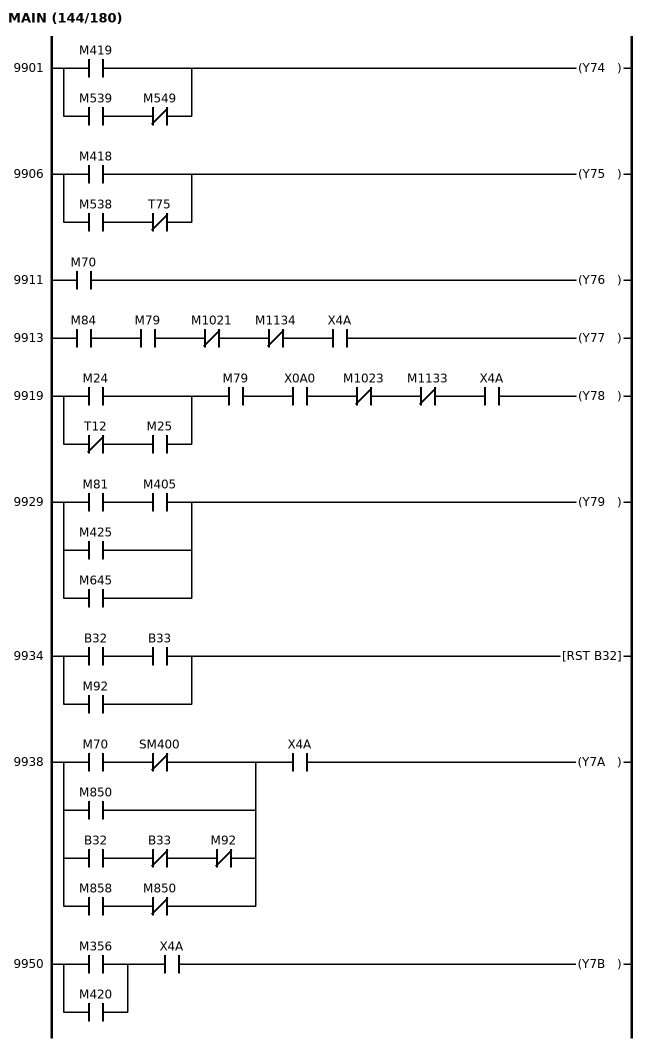
9901  LD      M419
      LD      M539
      ANI     M549
      ORB
      OUT     Y74
9906  LD      M418
      LD      M538
      ANI     T75
      ORB
      OUT     Y75
9911  LD      M70
      OUT     Y76
9913  LD      M84
      AND     M79
      ANI     M1021
      ANI     M1134
      AND     X4A
      OUT     Y77
9919  LD      M24
      LDI     T12
      AND     M25
      ORB
      AND     M79
      AND     X0A0
      ANI     M1023
      ANI     M1133
      AND     X4A
      OUT     Y78
9929  LD      M81
      AND     M405
      OR      M425
      OR      M645
      OUT     Y79
9934  LD      B32
      AND     B33
      OR      M92
      RST     B32
9938  LD      M70
      ANI     SM400
      OR      M850
      LD      B32
      ANI     B33
      ANI     M92
      ORB
      LD      M858
      ANI     M850
      ORB
      AND     X4A
      OUT     Y7A
9950  LD      M356
      OR      M420
      AND     X4A
      OUT     Y7B
